// TIA Portal V19 export
TYPE "LEXCHANGETRAY_typeSr1000ProfinetTelegram_operationResultStatus"
// stored: Access Published
   STRUCT
      statusBytes : Array[0..11] of Byte;
      readResultCode : UInt;
      presetResultCode : UInt;
      registerPresetDataResultCode : UInt;
      tuneResultCode : UInt;
      extReqResultCode : UInt;
      generalErrorCode : UInt;
   END_STRUCT;
END_TYPE
